// TIA Portal V16 export
// export: Created 2023-03-29T11:04:55.7817878Z, ExportSetting WithDefaults, DisplayName Totally Integrated Automation Portal, DisplayVersion V16 Update 6, DisplayName TIA Portal Version Control Interface, DisplayVersion V16 Update 2, DisplayName TIA Portal Openness, DisplayVersion V16 Update 6, DisplayName STEP 7 Professional, DisplayVersion V16 Update 6, DisplayName STEP 7 Safety, DisplayVersion V16, DisplayName WinCC Advanced, DisplayVersion V16 Update 6
DATA_BLOCK "MB_SERVER_DB_100"   // DB115
// stored: AutoNumber true, DBAccessibleFromOPCUA true, InstanceOfName MB_SERVER, OfSystemLibElement MB_SERVER, OfSystemLibVersion 3.1
"MB_SERVER"
   // VAR_INPUT
   //    DISCONNECT : Bool;
   //    CONNECT_ID : UInt;
   //    IP_PORT : UInt;
   // END_VAR
   // VAR_OUTPUT
   //    NDR : Bool;
   //    DR : Bool;
   //    ERROR : Bool;
   //    STATUS : Word;
   // END_VAR
   // VAR_IN_OUT
   //    MB_HOLD_REG : Variant;
   // END_VAR
   // VAR
   //    TCON_SFB { S7_SetPoint := 'True'} : TCON;
   //    TDISCON_SFB { S7_SetPoint := 'True'} : TDISCON;
   //    TSEND_SFB { S7_SetPoint := 'True'} : TSEND;
   //    TRCV_SFB { S7_SetPoint := 'True'} : TRCV;
   //    TCON_Param { S7_SetPoint := 'True'} : TCON_Param;
   //    MB_State : UInt;
   //    Request_Count : UInt;
   //    Server_Message_Count : UInt;
   //    Xmt_Rcv_Count : UInt;
   //    Exception_Count : UInt;
   //    Success_Count : UInt;
   //    SL_Status_Hold : UInt;
   //    HR_Start_Offset : UInt;
   //    Init_OK : Bool;
   //    SL_Error_State : Bool;
   //    Connected : Bool;
   //    XMT_Set_NDR : Bool;
   //    XMT_Set_DR : Bool;
   // END_VAR
BEGIN
END_DATA_BLOCK
